TYPE WRITE_PAR :
STRUCT
	WriteAddress: WORD;
	WriteQty: WORD;
	AuxArr : ARRAY[1..10] OF DINT;
	
	bBusy: BOOL;
	bError: BOOL;
	commTrig: R_TRIG;
END_STRUCT
END_TYPE

(* stored: Version 1.1.0.1, ProductVersion 3.1.4024.13
   DUT WRITE_PAR: Id {e100ebd4-4cda-48d9-8a64-0cf0f1f52c3c} *)
